// TIA Portal V20 export
DATA_BLOCK "Instance_FB_DataLog_DB"   // DB110
// stored: AutoNumber false, InstanceOfName FB_DataLog, InstanceOfType FB
"FB_DataLog"
   // VAR_INPUT
   //    DataLogCreate_REQ : Bool;
   //    DataLogOpen_REQ : Bool;
   //    DataLogWrite_REQ : Bool;
   //    DataLogClose_REQ : Bool;
   //    DataLogClear_REQ : Bool;
   //    DataLogDelete_REQ : Bool;
   // END_VAR
   // VAR_OUTPUT
   //    DataLogCreate_DONE : Bool;
   //    DataLogCreate_BUSY : Bool;
   //    DataLogCreate_ERROR : Bool;
   //    DataLogCreate_STATUS : Word;
   //    DataLogOpen_DONE : Bool;
   //    DataLogOpen_BUSY : Bool;
   //    DataLogOpen_ERROR : Bool;
   //    DataLogOpen_STATUS : Word;
   //    DataLogWrite_DONE : Bool;
   //    DataLogWrite_BUSY : Bool;
   //    DataLogWrite_ERROR : Bool;
   //    DataLogWrite_STATUS : Word;
   //    DataLogClose_DONE : Bool;
   //    DataLogClose_BUSY : Bool;
   //    DataLogClose_ERROR : Bool;
   //    DataLogClose_STATUS : Word;
   //    DataLogClear_DONE : Bool;
   //    DataLogClear_BUSY : Bool;
   //    DataLogClear_ERROR : Bool;
   //    DataLogClear_STATUS : Word;
   //    DataLogDelete_DONE : Bool;
   //    DataLogDelete_BUSY : Bool;
   //    DataLogDelete_ERROR : Bool;
   //    DataLogDelete_STATUS : Word;
   // END_VAR
   // VAR_IN_OUT
   //    ID : DWord;
   //    "NAME" : Variant;
   //    DataLogCreate_HEADER : Variant;
   //    DATA : Variant;
   // END_VAR
   // VAR
   //    Enable_DataLogOpen : Bool;
   //    Enable_DataLogWrite : Bool;
   //    Axiliar_P_Trig_0 : Bool;
   //    Axiliar_P_Trig_1 : Bool;
   //    Axiliar_P_Trig_2 : Bool;
   //    Axiliar_P_Trig_3 : Bool;
   //    Axiliar_P_Trig_4 : Bool;
   //    Axiliar_P_Trig_5 : Bool;
   //    Axiliar_P_Trig_6 : Bool;
   //    Axiliar_P_Trig_7 : Bool;
   //    Axiliar_P_Trig_8 : Bool;
   //    DataLogCreate_Instance { S7_SetPoint := 'True'} : DataLogCreate;
   //    DataLogOpen_Instance { S7_SetPoint := 'True'} : DataLogOpen;
   //    DataLogWrite_Instance { S7_SetPoint := 'True'} : DataLogWrite;
   //    DataLogClose_Instance { S7_SetPoint := 'True'} : DataLogClose;
   //    DataLogClear_Instance { S7_SetPoint := 'True'} : DataLogClear;
   //    DataLogDelete_Instance { S7_SetPoint := 'True'} : DataLogDelete;
   // END_VAR
BEGIN
END_DATA_BLOCK
